// TIA Portal project "N19-3001" (V15)

(* hardware
DEVICE "S71500/ET200MP station_1"  S7-1500 station
   slot 0: "Rail_0"  Rack  6ES7 590-1***0-0AA0
   slot 1: "PLC_1"  CPU 1513F-1 PN  6ES7 513-1FL02-0AB0  V2.5
      slot 3: "CPU display_1"  6ES7591-1AA00-0AA0
DEVICE "RH1"  ET 200SP-Station
   slot 0: "Rack_0"  Rack  6ES5 710-8MAx1
   slot 0: "RH1_cp200"  IM 155-6 PN ST  6ES7 155-6AU00-0BN0  V3.3
   slot 1: "cp201"  F-DI 8x24VDC HF  6ES7 136-6BA00-0CA0  V1.0
      slot 1: "cp201"  F-DI 8x24VDC HF
   slot 2: "cp202"  F-DI 8x24VDC HF  6ES7 136-6BA00-0CA0  V1.0
      slot 1: "cp202"  F-DI 8x24VDC HF
   slot 3: "cp203"  F-DQ 8x24VDC/0.5A PP HF  6ES7 136-6DC00-0CA0  V1.0
      slot 1: "cp203"  F-DQ 8x24VDC/0.5A PP HF
   slot 4: "cp204"  DI 16x24VDC ST  6ES7 131-6BH01-0BA0  V0.0
      slot 1: "cp204"  DI 16x24VDC ST
   slot 5: "cp205"  DI 16x24VDC ST  6ES7 131-6BH01-0BA0  V0.0
      slot 1: "cp205"  DI 16x24VDC ST
   slot 6: "cp206"  DI 16x24VDC ST  6ES7 131-6BH01-0BA0  V0.0
      slot 1: "cp206"  DI 16x24VDC ST
   slot 7: "cp207"  DI 16x24VDC ST  6ES7 131-6BH01-0BA0  V0.0
      slot 1: "cp207"  DI 16x24VDC ST
   slot 8: "cp208"  DI 16x24VDC ST  6ES7 131-6BH01-0BA0  V0.0
      slot 1: "cp208"  DI 16x24VDC ST
   slot 9: "cp209"  DI 16x24VDC ST  6ES7 131-6BH01-0BA0  V0.0
      slot 1: "cp209"  DI 16x24VDC ST
   slot 10: "cp210"  DI 16x24VDC ST  6ES7 131-6BH01-0BA0  V0.0
      slot 1: "cp210"  DI 16x24VDC ST
   slot 11: "cp211"  DI 16x24VDC ST  6ES7 131-6BH01-0BA0  V0.0
      slot 1: "cp211"  DI 16x24VDC ST
   slot 12: "cp212"  AI 8xRTD/TC 2-wire HF  6ES7 134-6JF00-0CA1  V2.0
      slot 1: "cp212"  AI 8xRTD/TC 2-wire HF
   slot 13: "cp213"  AI 8xRTD/TC 2-wire HF  6ES7 134-6JF00-0CA1  V2.0
      slot 1: "cp213"  AI 8xRTD/TC 2-wire HF
   slot 127: "BA 2xRJ45"  BA 2xRJ45  6ES7 193-6AR00-0AA0  V0.0
      slot 1: "Port_1"  X1 P1 R  6ES7 193-6AR00-0AA0  V0.0
      slot 2: "Port_2"  X1 P2 R  6ES7 193-6AR00-0AA0  V0.0
DEVICE "RM2"  ET 200SP-Station
   slot 0: "Rack_0"  Rack  6ES5 710-8MAx1
   slot 0: "RM2_cp400"  IM 155-6 PN ST  6ES7 155-6AU00-0BN0  V3.3
   slot 1: "pm401"  DQ 8x24VDC/0.5A ST  6ES7 132-6BF01-0BA0  V0.0
      slot 1: "pm401"  DQ 8x24VDC/0.5A ST
   slot 2: "pm402"  DQ 8x24VDC/0.5A ST  6ES7 132-6BF01-0BA0  V0.0
      slot 1: "pm402"  DQ 8x24VDC/0.5A ST
   slot 127: "BA 2xRJ45"  BA 2xRJ45  6ES7 193-6AR00-0AA0  V0.0
      slot 1: "Port_1"  X1 P1 R  6ES7 193-6AR00-0AA0  V0.0
      slot 2: "Port_2"  X1 P2 R  6ES7 193-6AR00-0AA0  V0.0
DEVICE "RK1"  ET 200SP-Station
   slot 0: "Rack_0"  Rack  6ES5 710-8MAx1
   slot 0: "RK1_cp300"  IM 155-6 PN ST  6ES7 155-6AU00-0BN0  V3.3
   slot 1: "cp301"  F-DI 8x24VDC HF  6ES7 136-6BA00-0CA0  V1.0
      slot 1: "cp301"  F-DI 8x24VDC HF
   slot 2: "cp302"  F-DI 8x24VDC HF  6ES7 136-6BA00-0CA0  V1.0
      slot 1: "cp302"  F-DI 8x24VDC HF
   slot 3: "F-DQ 4x24VDC/2A PM HF_1"  F-DQ 4x24VDC/2A PM HF  6ES7 136-6DB00-0CA0  V1.0
      slot 1: "F-DQ 4x24VDC/2A PM HF_1"  F-DQ 4x24VDC/2A PM HF
   slot 4: "cp304"  DQ 8x24VDC/0.5A ST  6ES7 132-6BF01-0BA0  V0.0
      slot 1: "cp304"  DQ 8x24VDC/0.5A ST
   slot 5: "cp305"  DQ 8x24VDC/0.5A ST  6ES7 132-6BF01-0BA0  V0.0
      slot 1: "cp305"  DQ 8x24VDC/0.5A ST
   slot 6: "cp306"  DQ 8x24VDC/0.5A ST  6ES7 132-6BF01-0BA0  V0.0
      slot 1: "cp306"  DQ 8x24VDC/0.5A ST
   slot 7: "cp307"  DQ 8x24VDC/0.5A ST  6ES7 132-6BF01-0BA0  V0.0
      slot 1: "cp307"  DQ 8x24VDC/0.5A ST
   slot 8: "cp308"  DQ 8x24VDC/0.5A ST  6ES7 132-6BF01-0BA0  V0.0
      slot 1: "cp308"  DQ 8x24VDC/0.5A ST
   slot 9: "cp309"  DQ 8x24VDC/0.5A ST  6ES7 132-6BF01-0BA0  V0.0
      slot 1: "cp309"  DQ 8x24VDC/0.5A ST
   slot 10: "cp310"  DQ 8x24VDC/0.5A ST  6ES7 132-6BF01-0BA0  V0.0
      slot 1: "cp310"  DQ 8x24VDC/0.5A ST
   slot 11: "cp311"  DQ 8x24VDC/0.5A ST  6ES7 132-6BF01-0BA0  V0.0
      slot 1: "cp311"  DQ 8x24VDC/0.5A ST
   slot 12: "cp312"  DQ 8x24VDC/0.5A ST  6ES7 132-6BF01-0BA0  V0.0
      slot 1: "cp312"  DQ 8x24VDC/0.5A ST
   slot 127: "BA 2xRJ45"  BA 2xRJ45  6ES7 193-6AR00-0AA0  V0.0
      slot 1: "Port_1"  X1 P1 R  6ES7 193-6AR00-0AA0  V0.0
      slot 2: "Port_2"  X1 P2 R  6ES7 193-6AR00-0AA0  V0.0
DEVICE "RK2"  ET 200SP-Station
   slot 0: "Rack_0"  Rack  6ES5 710-8MAx1
   slot 0: "RK2_cp400"  IM 155-6 PN ST  6ES7 155-6AU00-0BN0  V3.3
   slot 1: "cp400"  DI 8x24VDC ST  6ES7 131-6BF01-0BA0  V0.0
      slot 1: "cp400"  DI 8x24VDC ST
   slot 2: "cp401"  DI 8x24VDC ST  6ES7 131-6BF01-0BA0  V0.0
      slot 1: "cp401"  DI 8x24VDC ST
   slot 3: "cp402"  DI 8x24VDC ST  6ES7 131-6BF01-0BA0  V0.0
      slot 1: "cp402"  DI 8x24VDC ST
   slot 4: "cp403"  DI 8x24VDC ST  6ES7 131-6BF01-0BA0  V0.0
      slot 1: "cp403"  DI 8x24VDC ST
   slot 5: "cp404"  DI 8x24VDC ST  6ES7 131-6BF01-0BA0  V0.0
      slot 1: "cp404"  DI 8x24VDC ST
   slot 6: "cp405"  DI 8x24VDC ST  6ES7 131-6BF01-0BA0  V0.0
      slot 1: "cp405"  DI 8x24VDC ST
   slot 7: "cp406"  CM 4xIO-Link  6ES7 137-6BD00-0BA0  V2.2
      slot 1: "cp406"  6ES7 137-6BD00-0BA0
   slot 127: "BA 2xRJ45"  BA 2xRJ45  6ES7 193-6AR00-0AA0  V0.0
      slot 1: "Port_1"  X1 P1 R  6ES7 193-6AR00-0AA0  V0.0
      slot 2: "Port_2"  X1 P2 R  6ES7 193-6AR00-0AA0  V0.0
DEVICE "GF3"  GSD.Device.PN
   slot 0: "Rack"  Rack  V1.0
   slot 0: "GF3"  Schneider Electric Lexium 32  LXM32M
      slot 0: "Schneider Electric Lexium 32"  Schneider Electric Lexium 32
      slot 1: "X1"  X1
         slot 1: "Port 1"  Port 1
         slot 2: "Port 2"  Port 2
   slot 1: "Drive Profile Lexium 1_1"  Drive Profile Lexium 1
      slot 0: "Drive Profile Lexium 1"  Drive Profile Lexium 1
DEVICE "GF2"  GSD.Device.PN
   slot 0: "Rack"  Rack  V1.0
   slot 0: "GF2"  Schneider Electric Lexium 32  LXM32M
      slot 0: "Schneider Electric Lexium 32"  Schneider Electric Lexium 32
      slot 1: "X1"  X1
         slot 1: "Port 1"  Port 1
         slot 2: "Port 2"  Port 2
   slot 1: "Drive Profile Lexium 1_1"  Drive Profile Lexium 1
      slot 0: "Drive Profile Lexium 1"  Drive Profile Lexium 1
DEVICE "GF1"  GSD.Device.PN
   slot 0: "Rack"  Rack  V1.0
   slot 0: "GF1"  Schneider Electric Lexium 32  LXM32M
      slot 0: "Schneider Electric Lexium 32"  Schneider Electric Lexium 32
      slot 1: "X1"  X1
         slot 1: "Port 1"  Port 1
         slot 2: "Port 2"  Port 2
   slot 1: "Drive Profile Lexium 1_1"  Drive Profile Lexium 1
      slot 0: "Drive Profile Lexium 1"  Drive Profile Lexium 1
*)

// ===== PLC "PLC_1"  CPU 1513F-1 PN =====

DATA_BLOCK "Main_Safety_RTG1_DB"   // DB1, F_DB
{ S7_Optimized_Access := 'TRUE' }
NAME : FUSI
VERSION : 0.1
// stored: InstanceOfName Main_Safety_RTG1
"Main_Safety_RTG1"
BEGIN
END_DATA_BLOCK

FUNCTION_BLOCK "Main_Safety_RTG1"   // FB1, F_FBD
{ S7_Optimized_Access := 'TRUE' }
VERSION : 0.1
BEGIN
END_FUNCTION_BLOCK

ORGANIZATION_BLOCK "Main"   // OB1, LAD, ProgramCycle
TITLE = "Main Program Sweep (Cycle)"
{ S7_Optimized_Access := 'TRUE' }
VERSION : 0.1
   VAR_INPUT
      Initial_Call : Bool;   // Initial call of this OB
      Remanence : Bool;   // =True, if remanent data are available
   END_VAR
BEGIN
END_ORGANIZATION_BLOCK